SUBAPPLICATION NumericValue_TO_CLIENT_1_0_OPC (* VT-Eingabefeld (CInputNumber) - NUR bei echter Eingabe (NumericValue_PHYSA feuert on-commit) - ruft eine entfernte OPC-UA-Methode MIT dem eingegebenen REAL-Wert als Argument auf (CALL_METHOD, AR_CLIENT_1_0). Rueckweg (Anzeige des tatsaechlich wirksamen/bestaetigten Werts auf demselben VT-Feld) laeuft separat und unkritisch ueber einen normalen Subscribe (Q_NumericValue_PHYSA) - kein Zirkelbezug, kein Merge/Last-Writer-Wins noetig (nur EIN Aufrufer pro Methode auf der Empfaengerseite, serialisiert durch den Methodenaufruf selbst). *)
  (* Standard: 61499-2; Description: Copyright (c) 2026 Meisterschulen am Ostbahnhof This program and the accompanying materials are made available under the terms of the Eclipse Public License 2.0 which is available at https://www.eclipse.org/legal/epl-2.0/ SPDX-License-Identifier: EPL-2.0 *)
  (* Version 1.0, 2026-09-23, Franz Höpfinger, Meisterschulen am Ostbahnhof, initial implementation - Franz: 'man macht auf STG4 2 METHODEN, die werden aufgerufen: vom Web-Dashboard oder von VT1, und zwar nur wenn jemand was eingibt... der rueckweg laeuft ueber einen Subscribe und ist unkritisch'. Fuer Druck (B20) ZERO/SPAN-Referenzwerte fern der Sensor-Station eingebbar, ohne AR2/Web-Override-Merge-Komplexitaet und ohne 2-Quellen-Schreiben-Problem. *)
  (* Version 1.1, 2026-09-25, Franz Höpfinger, Meisterschulen am Ostbahnhof, Call-Baustein AR_CLIENT_1_0 -> AR_CLIENT_1_0_UNGATED (bestaetigter Review-Fund auf PR #267): AR_CLIENT_1_0's interner E_D_FF_ANY unterdrueckte eine erneute CALL_METHOD, wenn der neu eingegebene Wert zufaellig mit dem zuletzt gesendeten uebereinstimmte - dieses SubApp ruft aber laut Kommentar/Design 'NUR bei echter Eingabe', unabhaengig vom Wert. *)
  PACKAGE MyLib::sys;
  IMPORT isobus::UT::Q::const::IDs::ID_NULL;
  IMPORT logiBUS::utils::conversion::phys::NumericObjectPool_S;
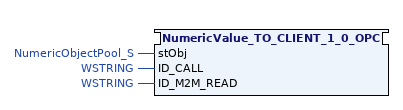
  VAR_INPUT
    stObj : logiBUS::utils::conversion::phys::NumericObjectPool_S := (u16ObjId := ID_NULL, r32Scale := 1.0, i32Offset := 0, u8Decimals := 1); (* Object ID + Scale/Offset/Decimals des VT-Eingabefelds (Ein- UND Ausgabe: bestaetigter Wert wird hier zurueckgeschrieben) *)
    ID_CALL : WSTRING; (* Remote-Methodenadresse (ACTION=CALL_METHOD) - wird NUR bei einer echten VT-Eingabe (NumericValue_PHYSA-Commit) mit dem eingegebenen Wert als Argument aufgerufen *)
    ID_M2M_READ : WSTRING; (* Remote-Subscribe-Adresse (REAL, ACTION=SUBSCRIBE) - liefert den tatsaechlich wirksamen/bestaetigten Wert zur Anzeige auf demselben VT-Feld zurueck (unkritischer Rueckweg, reines Lesen) *)
  END_VAR
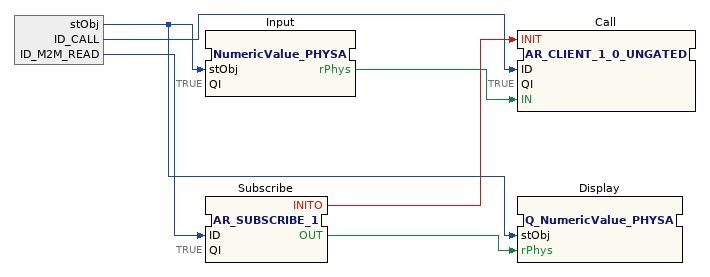
  FBS
    Input : isobus::UT::io::NumericValue::NumericValue_PHYSA(QI := TRUE);
    Call : adapter::net::AR_CLIENT_1_0_UNGATED(QI := TRUE);
    Subscribe : adapter::net::AR_SUBSCRIBE_1(QI := TRUE);
    Display : isobus::UT::Q::Q_NumericValue_PHYSA;
  END_FBS
  EVENT_CONNECTIONS
    Subscribe.INITO TO Call.INIT;
  END_CONNECTIONS
  DATA_CONNECTIONS
    stObj TO Input.stObj;
    stObj TO Display.stObj;
    ID_CALL TO Call.ID;
    ID_M2M_READ TO Subscribe.ID;
  END_CONNECTIONS
  ADAPTER_CONNECTIONS
    Input.rPhys TO Call.IN;
    Subscribe.OUT TO Display.rPhys;
  END_CONNECTIONS
END_SUBAPPLICATION
